RoboDK station: Seguir_Trayectoria_2.rdk

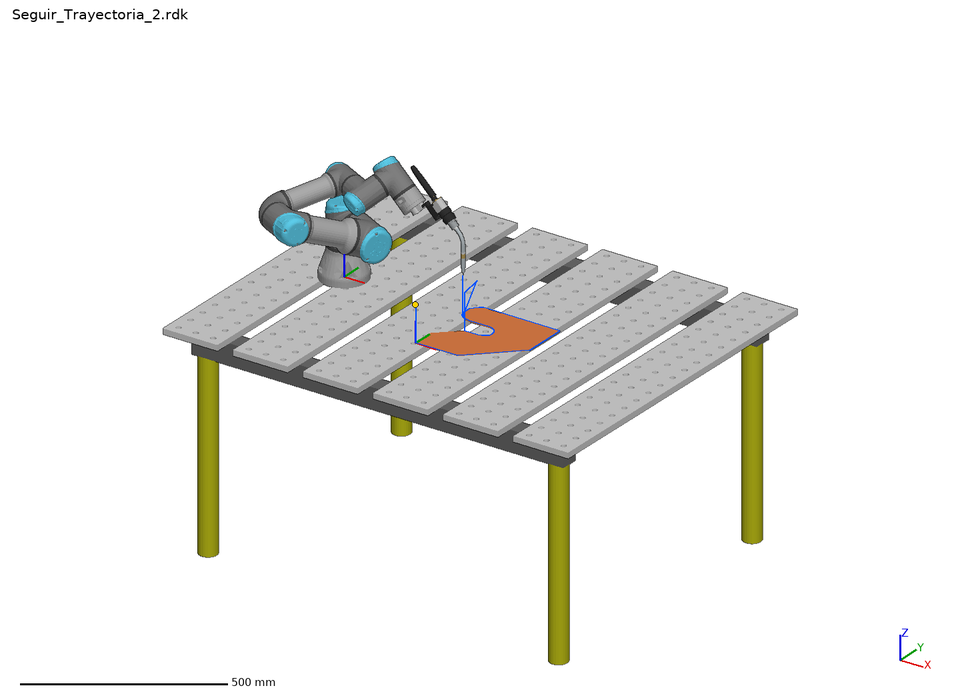
[picture v0: the station drawn from its stored meshes, robots at their saved joint values, targets as dots, program paths as lines]
Station Seguir_Trayectoria_2 (saved by RoboDK 5.7.3). Poses are relative to the parent item; angles as X-Y-Z fixed-axis rotations.
  - frame UR3e Base at (-400, 0, 0) mm
    - robot UR3e: 6 axes, payload 3 kg, reach 500 mm, repeatability 0.03 mm, weight 11 kg
        modified DH rows (alpha deg, a mm, theta deg, d mm): 0, 0, 0, 151.9; 90, 0, 180, 0; 0, 243.55, 0, 0; 0, 213.2, 0, 131.05; -90, 0, 0, 85.35; 90, 0, 180, 92.1
        joint limits [-360, -360, -360, -360, -360, -360] to [360, 360, 360, 360, 360, 360]; home [0, -90, -90, 0, 90, 0]; saved at [63.375, -22.155, -149.129, -74.577, 50.793, 144.665]
      - tool OTC Daihen FD-84 Welding Gun, TCP at (1, 0, 201) mm, rotated rx 0 ry 45 rz 0 deg, size 100.8 x 32.5 x 283.9 mm
  - object Table 1200x1000mm (Welding) at (0, 0, 0) mm, size 1193.8 x 965.2 x 609.6 mm, geometry from Table-1200x1000mm-Welding.sld
  - frame ref_objeto at (-50, -200, 0) mm
    - object Cutting sheet at (0, 0, 0) mm, size 250 x 250 x 3 mm, geometry from Cutting sheet.STEP
  - machining project Path1 ajustes: rotZ(0) | rotX(0)*rotY(0) | rotz(0) | onStart | onPathStart | onApproach | onPoint | onRetract | onFinish | SetRPM(%1) | SetTool(%1) | Extruder(%1) | default | default | OutOnMov(%1) | OutOffMov(%1) | onPathFinish | M_RunCode(%1)
  - program Path1 (52 instructions, listed below)
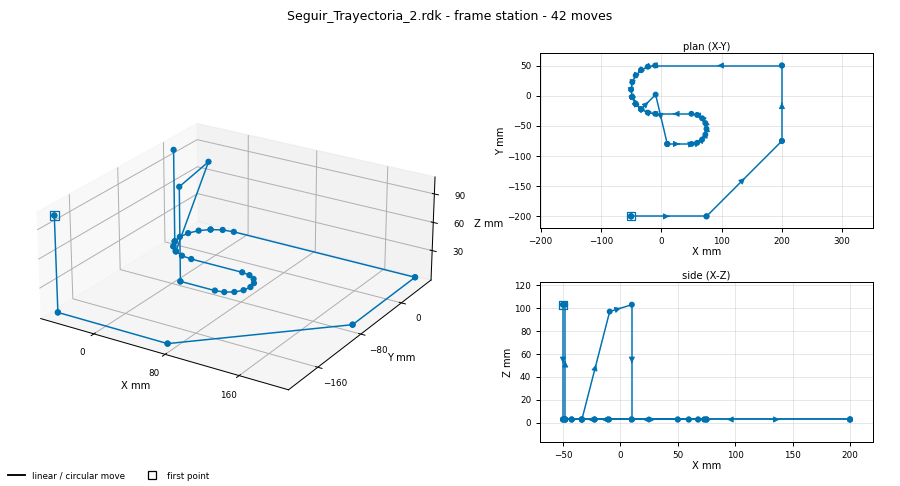
[picture p0: tool path of Seguir_Trayectoria_2.rdk in frame station, 42 of 42 moves have a stored position in this frame; points joined in program order, loops and branches not executed]

--- program Path1 (robot UR3e) ---
  Suave(1)
  Establecer velocidad (1000.0 mm/s)
  Est. Ref.: ref_objeto
  Est. herr: OTC Daihen FD-84 Welding Gun
  Mostrar OTC Daihen FD-84 Welding Gun
  MoveJ 1 to (0, 0, 103) mm, rotated rx -180 ry 0 rz -180 deg; joints [-22.178, -86.892, -134.914, -5.394, 105.481, 73.92]
  MoveL 2 to (0, 0, 103) mm, rotated rx -180 ry 0 rz -180 deg; joints [-22.178, -86.892, -134.914, -5.394, 105.481, 73.92]
  MoveL 3 to (0, 0, 3) mm, rotated rx -180 ry 0 rz -180 deg; joints [-22.178, -119.213, -143.552, 35.566, 105.481, 73.92]
  MoveL 4 to (0, 0, 3) mm, rotated rx -180 ry 0 rz -180 deg; joints [-22.178, -119.213, -143.552, 35.566, 105.481, 73.92]
  Establecer velocidad (50.0 mm/s)
  MoveL 5 to (125, 0, 3) mm, rotated rx -180 ry 0 rz -180 deg; joints [-13.64, -128.564, -114.971, 17.715, 99.599, 80.263]
  MoveL 6 to (125, 0, 3) mm, rotated rx -90 ry 0 rz -135 deg; joints [-18.488, -184.986, -86.9, 91.885, 108.488, 0]
  MoveL 7 to (250, 125, 3) mm, rotated rx -90 ry 0 rz -135 deg; joints [10.97, -186.095, -71.709, 77.805, 79.03, 0]
  MoveL 8 to (250, 125, 3) mm, rotated rx 180 ry 0 rz 180 deg; joints [8.306, -138.08, -92.074, 4.851, 84.137, 95.894]
  MoveL 9 to (250, 250, 3) mm, rotated rx -180 ry 0 rz 180 deg; joints [26.536, -136.45, -94.535, 2.802, 71.584, 109.449]
  MoveL 10 to (250, 250, 3) mm, rotated rx -180 ry 0 rz 180 deg; joints [26.536, -136.45, -94.535, 2.802, 71.584, 109.449]
  MoveL 11 to (40, 250, 3) mm, rotated rx -180 ry 0 rz -180 deg; joints [58.813, -107.089, -165.488, 29.954, 52.777, 139.435]
  MoveL 12 to (27.64, 248.04, 3) mm, rotated rx 180 ry 0 rz 180 deg; joints [63.198, -103.708, -170.459, 28.438, 50.866, 144.457]
  MoveL 13 to (16.49, 242.36, 3) mm, rotated rx -180 ry 0 rz 180 deg; joints [67.211, -98.327, -175.399, 24.899, 49.314, 149.283]
  MoveL 14 to (16.49, 242.36, 3) mm, rotated rx -180 ry 0 rz 180 deg; joints [67.211, -98.327, -175.399, 24.899, 49.314, 149.283]
  MoveL 15 to (7.64, 233.51, 3) mm, rotated rx 180 ry 0 rz 180 deg; joints [70.367, -75.775, -177.523, 1.87, 48.241, 153.229]
  MoveL 16 to (1.96, 222.36, 3) mm, rotated rx 180 ry 0 rz -180 deg; joints [71.711, -35.133, -174.883, -42.562, 47.826, 154.949]
  MoveL 17 to (0, 210, 3) mm, rotated rx 180 ry 0 rz -180 deg; joints [69.676, -21.683, -174.362, -54.801, 48.464, 152.354]
  MoveL 18 to (1.96, 197.64, 3) mm, rotated rx 180 ry 0 rz 160 deg; joints [73.023, -56.104, -164.446, -52.468, 45.08, 184.271]
  MoveL 19 to (1.96, 197.64, 3) mm, rotated rx 180 ry 0 rz 160 deg; joints [73.023, -56.104, -164.446, -52.468, 45.08, 184.271]
  MoveL 20 to (7.64, 186.49, 3) mm, rotated rx 180 ry 0 rz 160 deg; joints [68.409, -61.722, -166.02, -40.667, 45.022, 177.75]
  MoveL 21 to (16.49, 177.64, 3) mm, rotated rx -165.14 ry -13.55 rz 176.45 deg; joints [47.113, -80.077, -150.393, -26.374, 58.479, 129.362]
  Establecer velocidad (1000.0 mm/s)
  MoveL 22 to (16.49, 177.64, 3) mm, rotated rx -165.14 ry -13.55 rz 176.45 deg; joints [47.113, -80.077, -150.393, -26.374, 58.479, 129.362]
  MoveL 23 to (40.67, 201.82, 96.97) mm, rotated rx -165.14 ry -13.55 rz 176.45 deg; joints [46.771, -72.051, -125.011, -59.577, 58.558, 128.972]
  Establecer velocidad (1000.0 mm/s)
  MoveL 24 to (60, 120, 103) mm, rotated rx 180 ry 0 rz 180 deg; joints [15.365, -78.59, -142.072, -5.381, 79.201, 100.996]
  MoveL 25 to (60, 120, 3) mm, rotated rx 180 ry 0 rz 180 deg; joints [15.365, -119.023, -152.218, 45.198, 79.201, 100.996]
  MoveL 26 to (60, 120, 3) mm, rotated rx 180 ry 0 rz 180 deg; joints [15.365, -119.023, -152.218, 45.198, 79.201, 100.996]
  Establecer velocidad (50.0 mm/s)
  MoveL 27 to (100, 120, 3) mm, rotated rx -180 ry 0 rz -180 deg; joints [12.566, -120.567, -139.907, 34.78, 81.151, 98.957]
  MoveL 28 to (109.57, 121.9, 3) mm, rotated rx -180 ry 0 rz -180 deg; joints [12.51, -121.213, -137.203, 32.728, 81.189, 98.917]
  MoveL 29 to (117.68, 127.32, 3) mm, rotated rx -180 ry 0 rz -180 deg; joints [13.36, -121.692, -135.256, 31.162, 80.596, 99.533]
  MoveL 30 to (123.1, 135.43, 3) mm, rotated rx -180 ry 0 rz -180 deg; joints [14.927, -121.889, -134.303, 30.209, 79.505, 100.675]
  MoveL 31 to (125, 145, 3) mm, rotated rx -180 ry 0 rz 180 deg; joints [16.992, -121.743, -134.46, 29.925, 78.075, 102.193]
  MoveL 32 to (123.1, 154.57, 3) mm, rotated rx -180 ry 0 rz -180 deg; joints [19.317, -121.259, -135.713, 30.313, 76.473, 103.921]
  MoveL 33 to (117.68, 162.68, 3) mm, rotated rx 180 ry 0 rz 180 deg; joints [21.655, -120.512, -137.919, 31.336, 74.875, 105.682]
  MoveL 34 to (109.57, 168.1, 3) mm, rotated rx -180 ry 0 rz 180 deg; joints [23.736, -119.642, -140.809, 32.923, 73.464, 107.272]
  MoveL 35 to (100, 170, 3) mm, rotated rx -180 ry 0 rz 180 deg; joints [25.268, -118.837, -144.001, 34.961, 72.432, 108.457]
  MoveL 36 to (40, 170, 3) mm, rotated rx -180 ry 0 rz -180 deg; joints [35.541, -120.048, -165.268, 54.451, 65.73, 116.8]
  MoveL 37 to (27.64, 171.96, 3) mm, rotated rx 180 ry 0 rz -180 deg; joints [39.793, -126.389, -171.175, 65.101, 63.092, 120.498]
  MoveL 38 to (16.49, 177.64, 3) mm, rotated rx -180 ry 0 rz 160 deg; joints [62.699, -73.954, -166.656, -22.148, 45.463, 169.73]
  MoveL 39 to (7.64, 186.49, 3) mm, rotated rx 180 ry 0 rz 160 deg; joints [68.409, -61.722, -166.02, -40.667, 45.022, 177.75]
  MoveL 40 to (1.96, 197.64, 3) mm, rotated rx 180 ry 0 rz 160 deg; joints [73.023, -56.104, -164.446, -52.468, 45.08, 184.271]
  Establecer velocidad (1000.0 mm/s)
  MoveL 41 to (1.96, 197.64, 3) mm, rotated rx 180 ry 0 rz 160 deg; joints [73.023, -56.104, -164.446, -52.468, 45.08, 184.271]
  MoveL 42 to (1.96, 197.64, 103) mm, rotated rx 180 ry 0 rz 180 deg; joints [63.375, -22.155, -149.129, -74.577, 50.793, 144.665]
